// TIA Portal V20 export
FUNCTION_BLOCK "LER_EQP_m_Interface"   // FB197, LAD
// stored: Access Published, MemoryReserve 100, SetENOAutomatically false
   VAR_INPUT
      enable : Bool;
      heartBeat : Byte;
      unitStatus : "LAF_typeUnitStatus";
      unitAlarms : "LAF_typeAlarms";
      partData : "LER_typePartData";
   END_VAR
   VAR_IN_OUT
      LOGSCommunication : "LER_type_mzc_Communication";
      configuration : "LER_typeCommunicationConfiguration";
      moduleInterface : "LER_typeCommunicationInterface";
      controlNode : "LER_typeCommunicationControlNode";
   END_VAR
   VAR
      instEQP_Interface_Communication { S7_SetPoint := 'True'} : "LER_EQP_m_Communication";
   END_VAR
BEGIN

REGION Network 2: EQP Interface Communication ReelCut <-> Stack
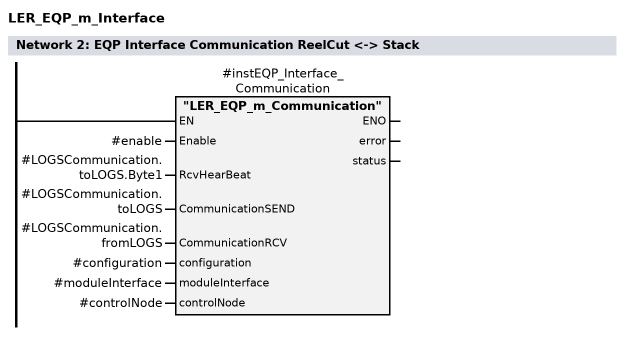
   RUNG wire#powerrail
      #instEQP_Interface_Communication(Enable := #enable, RcvHearBeat := #LOGSCommunication.toLOGS.Byte1, CommunicationSEND := #LOGSCommunication.toLOGS, CommunicationRCV := #LOGSCommunication.fromLOGS, configuration := #configuration, moduleInterface := #moduleInterface, controlNode := #controlNode, error =>, status =>)
   END_RUNG
   // the same network as SCL:
   #instEQP_Interface_Communication(Enable := #enable,   // "LER_EQP_m_Communication"
                           RcvHearBeat := #LOGSCommunication.toLOGS.Byte1,
                           CommunicationSEND := #LOGSCommunication.toLOGS,
                           CommunicationRCV := #LOGSCommunication.fromLOGS,
                           configuration := #configuration,
                           moduleInterface := #moduleInterface,
                           controlNode := #controlNode);
END_REGION
END_FUNCTION_BLOCK
